TYPE AX5000_S_0043 :
STRUCT
	Velocity_polarity_parameter:UINT;
END_STRUCT
END_TYPE

(* stored: Version 1.1.0.1, ProductVersion 3.1.4024.3
   DUT AX5000_S_0043: Id {31a13321-0c93-4230-8a77-d4c230e4a293} *)
